{attribute 'qualified_only'}
VAR_GLOBAL
	flSS1				: FB_BaseFlag;
	flSTO				: FB_BaseFlag;
	
END_VAR

(* stored: Version 1.1.0.1
   GVL GVL_MCSafety: Id {451bd6aa-b1ce-4028-9df3-f0fda13e64ea} *)
